(*

short summary
=============

.. <legal notes>

legal notes
=================
| SPDX-FileCopyrightText: © 2023 ekvip automation GmbH <info@ekvip.de>
| SPDX-License-Identifier: Apache-2.0
| For details check: Apache-2.0_

.. _Apache-2.0: https://www.apache.org/licenses/LICENSE-2.0

.. </legal notes>

*)

{warning 'header is generated please add your documentation'}
INTERFACE IInt EXTENDS CNM_AbstractObject.IObject

(*

short summary
=============

.. <legal notes>

legal notes
=================
| SPDX-FileCopyrightText: © 2023 ekvip automation GmbH <info@ekvip.de>
| SPDX-License-Identifier: Apache-2.0
| For details check: Apache-2.0_

.. _Apache-2.0: https://www.apache.org/licenses/LICENSE-2.0

.. </legal notes>

*)

{warning 'header is generated please add your documentation'}
PROPERTY value : INT
GET
END_GET
SET
END_SET
END_PROPERTY

END_INTERFACE

(* stored: Version 1.1.0.1, ProductVersion 3.1.4024.12
   Itf IInt: Id {abaa5336-5f86-4fb9-aee6-d20b6985e7be}
   Property value: Id {907a7302-4458-4409-9e80-21fdf1b61bd0}
   Get Get: Id {0a4b1468-d3b4-4ccc-b59b-cbb9260cd6d2}
   Set Set: Id {4a8e0d2d-53f2-4e04-aea1-9ad6e61ac496} *)
